// This function has been automatically generated from the project information.
{attribute 'signature_flag' := '1073741824'}
{attribute 'TcGenerated'}
{attribute 'no-analysis'}
FUNCTION F_GetCompany : WSTRING
VAR_INPUT
	
END_VAR

F_GetCompany := "BeckhoffUK";

END_FUNCTION

(* stored: Version 1.1.0.1
   POU F_GetCompany: Id {d383df96-6c93-4ff2-bb0d-d212d2c00da1}, SpecialFunc None *)
